TYPE ST_ChEp1PrepareWaferTransferParam :
STRUCT
END_STRUCT
END_TYPE

(* stored: Version 1.1.0.1, ProductVersion 3.1.4026.18
   DUT ST_ChEp1PrepareWaferTransferParam: Id {b5a49ec2-cb1f-427e-897c-e69acfb39fec} *)
